DATA_BLOCK "DB_SSM_Type"
TITLE =%version: 0.08 % CN: 20
//History:
//This version  %created_by: nljsla %
//              %date_created: Monday, February 06, 2017 4:27:08 PM %
//              %release: VI_GEN/RA_Dev %
//
//Modification History:                                   By:    Date:     Rev:
//----------------------------------------------------  -------  --------  -----
//ra#20472: Due to SSM master/slave added link error    nljsla   06-02-17   0.08
//ra#16735: DI NON_RETAIN PLC Memory                    nlHdL    13-12-16   0.07
//ra#16493: Update DB_SSM_Type after stopped ext        nlHdL    05-09-16   0.06
//ra#16493: Update DB_SSM_Type after stopped_ext        nlHdL    05-09-16   0.06
//ra#9751: Add source files ECS-P to VI_RAW             nlHdL    14-12-15   0.05
//ra#9751: Add source files ECS-P to VI_RAW             nlHdL    07-12-15   0.05
//7324: ECS-P General from the RD to RA for platform    nlHdL    06-07-15   0.05
//17046: Ready to Restart not visible on HMI or SCADA   nlHdL    30-04-15   0.05
//17783: Started is Bit 13 in Overall Status            nlHdL    10-02-14   0.04
//15797: Keyword release added                          nlwwij   26-09-13   0.03
//CR5712 Not used errors have number -1                 nlHdL    24-09-10   0.02
//Initial Revision                                      nlMRe    22-09-10   0.01
//
FAMILY : General
VERSION : 0.0
NON_RETAIN


  STRUCT
   Type_Component : BYTE ;	//Type of the component (1 = Section, 0 = Other)
   Record_Length : BYTE ;	//Number of the Detailed Status in the UDT
   Status : ARRAY  [1 .. 16 ] OF "UDT_Comp_Status";
  END_STRUCT ;
BEGIN
   Type_Component := B#16#0;
   Record_Length := B#16#16;
   Status[1].HMI_Text_Number := -1;
   Status[1].Overall_Status_Relation := B#16#13;
   Status[1].General_Status_Relation := B#16#13;
   Status[2].HMI_Text_Number := -1;
   Status[2].Overall_Status_Relation := B#16#8;
   Status[2].General_Status_Relation := B#16#9;
   Status[3].HMI_Text_Number := -1;
   Status[3].Overall_Status_Relation := B#16#6;
   Status[3].General_Status_Relation := B#16#7;
   Status[4].HMI_Text_Number := -1;
   Status[4].Overall_Status_Relation := B#16#7;
   Status[4].General_Status_Relation := B#16#8;
   Status[5].HMI_Text_Number := -1;
   Status[5].Overall_Status_Relation := B#16#5;
   Status[5].General_Status_Relation := B#16#4;
   Status[6].HMI_Text_Number := -1;
   Status[6].Overall_Status_Relation := B#16#0;
   Status[6].General_Status_Relation := B#16#0;
   Status[7].HMI_Text_Number := -1;
   Status[7].Overall_Status_Relation := B#16#0;
   Status[7].General_Status_Relation := B#16#0;
   Status[8].HMI_Text_Number := -1;
   Status[8].Overall_Status_Relation := B#16#0;
   Status[8].General_Status_Relation := B#16#0;
   Status[9].HMI_Text_Number := 54;
   Status[9].Overall_Status_Relation := B#16#4;
   Status[9].General_Status_Relation := B#16#3;
   Status[10].HMI_Text_Number := -1;
   Status[10].Overall_Status_Relation := B#16#0;
   Status[10].General_Status_Relation := B#16#0;
   Status[11].HMI_Text_Number := -1;
   Status[11].Overall_Status_Relation := B#16#0;
   Status[11].General_Status_Relation := B#16#0;
   Status[12].HMI_Text_Number := -1;
   Status[12].Overall_Status_Relation := B#16#0;
   Status[12].General_Status_Relation := B#16#0;
   Status[13].HMI_Text_Number := -1;
   Status[13].Overall_Status_Relation := B#16#0;
   Status[13].General_Status_Relation := B#16#0;
   Status[14].HMI_Text_Number := -1;
   Status[14].Overall_Status_Relation := B#16#0;
   Status[14].General_Status_Relation := B#16#0;
   Status[15].HMI_Text_Number := -1;
   Status[15].Overall_Status_Relation := B#16#0;
   Status[15].General_Status_Relation := B#16#0;
   Status[16].HMI_Text_Number := -1;
   Status[16].Overall_Status_Relation := B#16#0;
   Status[16].General_Status_Relation := B#16#0;
END_DATA_BLOCK

